// Phase 0 - E_LMH
// Rev 1.0 - March 14, 2024

TYPE E_LMH :
(
	eLow			 													:= 0,
	eMid,
	eHigh
);
END_TYPE

(* stored: Version 1.1.0.1, ProductVersion 3.1.4024.12
   DUT E_LMH: Id {9f47d9bd-4b97-49c2-bfd1-fce29d03bc1d} *)
